{attribute 'qualified_only'}
{attribute 'strict'}
TYPE eTransitionType :
(
	None 		:=	 0,
	Linear 		:=	 1,
	Exponential :=	 2,
	S_Type 		:=	 3
);
END_TYPE

(* stored: Version 1.1.0.1, ProductVersion 3.1.4024.5
   DUT eTransitionType: Id {61935f21-fa84-4566-a236-09c8f4c122e1} *)
